Yaskawa INFORM job: TEST2.JBI

/JOB
//NAME TEST2
//POS
///NPOS 1,1,0,0,0,0
///TOOL 0
///POSTYPE ROBOT
///RECTAN
///RCONF 0,0,0,0,0,0,0,0,0,0,0,0,0,0,0,0,0,0,0,0,0,0,0,0
C00000=778.900,274.659,-1127.102,1.1211,49.7689,-139.7600
BC00000=1011.689,4837.660,450.146
//INST
///DATE 2024/01/25 09:44
///ATTR SC,RW,RJ
////FRAME ROBOT
///GROUP1 RB1,BS1
NOP
MOVJ C00000 BC00000 VJ=0.78
END
